FUNCTION_BLOCK HardeningProcess
VAR_INPUT
	MethodCall : BOOL;
	InputSensor: BOOL;
	HardeningTime : TIME;
	NotAusSignal : BOOL;
	AutomaticMode: BOOL;
END_VAR
VAR_OUTPUT
	HardeningProcess : BOOL;
END_VAR
VAR
//FlipFlop
	RS_HardeningProcess: RS;
//Zeitverzögerung
	TOF_HardeningTime: TOF;
//Flanke	
	R_TRIG_MethodCall: R_TRIG;
END_VAR
VAR // added by the converter: edge detectors and wires of the graphical bodies
    _w1 : BOOL;
END_VAR

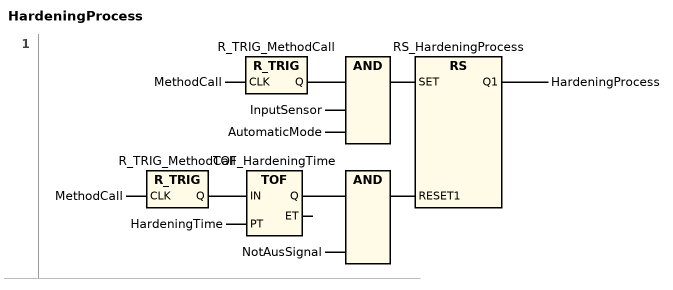
// NETWORK 1
R_TRIG_MethodCall(CLK := MethodCall); // R_TRIG
_w1 := R_TRIG_MethodCall.Q AND InputSensor AND AutomaticMode;
R_TRIG_MethodCall(CLK := MethodCall); // R_TRIG
TOF_HardeningTime(IN := R_TRIG_MethodCall.Q, PT := HardeningTime); // TOF
RS_HardeningProcess(SET := _w1, RESET1 := TOF_HardeningTime.Q AND NotAusSignal); // RS
HardeningProcess := RS_HardeningProcess.Q1;

END_FUNCTION_BLOCK

(* stored: Version 1.1.0.1, ProductVersion 3.1.4024.15
   POU HardeningProcess: Id {9bd305b2-8722-4353-b94b-a4a695281d20}, SpecialFunc None *)
